{attribute 'hide'}
FUNCTION_BLOCK PUBLIC Mock_FileSystemEntry EXTENDS FileSystemEntry

END_FUNCTION_BLOCK

(* stored: Version 1.1.0.1, ProductVersion 3.1.4024.9
   POU Mock_FileSystemEntry: Id {acbcab05-a2a1-47d3-8447-d5538d9585da}, SpecialFunc None *)
